// TIA Portal V19 export
FUNCTION "FC_FW_Auftrag_Step5_NB" : Void   // FC185, LAD
TITLE = Schritt CM04 -> WR02
{ S7_Optimized_Access := 'TRUE' }
// Ältesten Warenträger in CM04 suchen und nach WR02 transportieren
// stored: AutoNumber false, SetENOAutomatically false
   VAR_INPUT
      Frg_Schritt : Bool;
   END_VAR
   VAR_OUTPUT
      nextStep : Bool;
      startStep : Bool;
      parkStep : Bool;
   END_VAR
   VAR_IN_OUT
      Quelle : Int;
      Ziel : Int;
      Positionen : Array[1..30] of "UDT_Auftrag_Pos";
      Frg_Ausfahrt : Bool;
   END_VAR
   VAR_TEMP
      Sperre_Kurz_li : Bool;
      Sperre_Kurz_re : Bool;
      Sperre_Lang : Bool;
      Vorzug : Bool;
      Befehl_ok : Bool;
      tmpQuelle : Int;
      Oldest : Real;
   END_VAR
BEGIN

REGION Network 1 (SCL)
   IF (#Quelle <> 0) AND (#Ziel <> 0) THEN
       #nextStep := #Positionen[#Quelle].Sperre;
       #startStep := NOT #nextStep;
       #Quelle := 0;
       #Ziel := 0;
       #Frg_Ausfahrt := NOT #startStep;
       RETURN;
   END_IF;

   #Quelle := 0;
   #Ziel := 0;
   #nextStep := FALSE;
   #startStep := FALSE;
END_REGION

REGION Network 2 (SCL): Anmeldung Großoptik
   //alle Positionen suchbar
   #Positionen[19].CheckSperre := FALSE;
   #Positionen[20].CheckSperre := FALSE;
   #Positionen[21].CheckSperre := FALSE;
   #Positionen[22].CheckSperre := FALSE;
   #Positionen[23].CheckSperre := FALSE;
   #Positionen[24].CheckSperre := FALSE;

   //
   #Oldest := 0;
   #tmpQuelle := 0;

   //CM04
   "FC_FW_Auftrag_Suche"(Pos1 := 19,
                         Pos2 := 24,
                         Positionen := #Positionen,
                         Quelle := #tmpQuelle,
                         Oldest := #Oldest);

   IF ((#tmpQuelle = 21) OR (#tmpQuelle = 22)) AND #Frg_Ausfahrt AND #Frg_Schritt THEN
       //Großoptik ist ältester
       #Vorzug := NOT "DI_QF_WR02_03".In.Req_Ausfahrt_GO;
       "DI_QF_WR02_03".In.Req_Ausfahrt_GO := TRUE;
   ELSE
       #Vorzug := FALSE;
       "DI_QF_WR02_03".In.Req_Ausfahrt_GO := FALSE;
   END_IF;

   IF (#tmpQuelle = 0) OR NOT #Frg_Schritt THEN
       #Frg_Ausfahrt := FALSE;
   END_IF;
END_REGION

REGION Network 3 (SCL): Positionen sperren
   IF NOT #Frg_Ausfahrt OR NOT #Frg_Schritt THEN
       #nextStep := TRUE;
       RETURN;
   END_IF;

   //Groß links nicht möglich
   #Positionen[21].CheckSperre := #Positionen[27].Sperre;

   //Groß rechts nicht möglich
   #Positionen[22].CheckSperre := #Positionen[28].Sperre;

   //kein Platz für Kurz links in WR02
   #Sperre_Kurz_li := (#Positionen[25].Sperre AND #Positionen[29].Sperre) OR #Vorzug;

   //kein Platz für Kurz rechts in WR02
   #Sperre_Kurz_re := (#Positionen[26].Sperre AND #Positionen[30].Sperre) OR #Vorzug;

   //kein Platz für Lang in WR02
   #Sperre_Lang := ((#Positionen[25].Sperre OR #Positionen[26].Sperre) AND (#Positionen[29].Sperre OR #Positionen[30].Sperre)) OR #Vorzug;

   //Lang in P19 oder
   //kein Platz auf rechter Seite
   //-> P20 sperren
   #Positionen[20].CheckSperre := #Sperre_Kurz_re OR (#Positionen[19].Wt_Typ = "WT_Typ_LS");

   //Lang in P19 und kein Platz für Lang oder
   //kein Platz auf linker Seite
   //-> P19 sperren
   #Positionen[19].CheckSperre := #Sperre_Kurz_li OR ((#Positionen[19].Wt_Typ = "WT_Typ_LS") AND #Sperre_Lang);

   //Lang in P23 oder
   //kein Platz auf rechter Seite
   //-> P24 sperren
   #Positionen[24].CheckSperre := #Sperre_Kurz_re OR (#Positionen[23].Wt_Typ = "WT_Typ_LS");

   //Lang in P23 und kein Platz für Lang oder
   //kein Platz auf linker Seite
   //-> P23 sperren
   #Positionen[23].CheckSperre := #Sperre_Kurz_li OR ((#Positionen[23].Wt_Typ = "WT_Typ_LS") AND #Sperre_Lang);
END_REGION

REGION Network 4 (SCL): Ältesten WT suchen
   //
   #Oldest := 0;
   #tmpQuelle := 0;

   //CM04
   "FC_FW_Auftrag_Suche"(Pos1 := 19,
                         Pos2 := 24,
                         Positionen := #Positionen,
                         Quelle := #tmpQuelle,
                         Oldest := #Oldest);
END_REGION

REGION Network 5 (SCL): Auswertung
   IF #tmpQuelle = 0 THEN
       //kein WT
       #nextStep := TRUE;
       RETURN;
   END_IF;

   IF NOT #Positionen[#tmpQuelle].Fertig THEN
       #parkStep := TRUE;
       RETURN;
   END_IF;

   IF (#tmpQuelle = 21) THEN
       //Gross links
       IF NOT #Positionen[27].Sperre THEN
           "FC_FW_Auftrag_Befehl"(inQuelle := #tmpQuelle,
                                  inZiel := 27,
                                  Befehl_ok => #Befehl_ok,
                                  outQuelle => #Quelle,
                                  outZiel => #Ziel);

           #nextStep := NOT #Befehl_ok;
       ELSE
           #nextStep := TRUE;
       END_IF;
       RETURN;
   END_IF;

   IF (#tmpQuelle = 22) THEN
       //Gross rechts
       IF NOT #Positionen[28].Sperre THEN
           "FC_FW_Auftrag_Befehl"(inQuelle := #tmpQuelle,
                                  inZiel := 28,
                                  Befehl_ok => #Befehl_ok,
                                  outQuelle => #Quelle,
                                  outZiel => #Ziel);

           #nextStep := NOT #Befehl_ok;
       ELSE
           #nextStep := TRUE;
       END_IF;
       RETURN;
   END_IF;

   IF (#Positionen[#tmpQuelle].Wt_Typ = "WT_Typ_LS") AND ((#tmpQuelle = 19) OR (#tmpQuelle = 23)) THEN
       //Lang
       IF NOT #Positionen[25].Sperre AND NOT #Positionen[26].Sperre THEN
           "FC_FW_Auftrag_Befehl"(inQuelle := #tmpQuelle,
                                  inZiel := 25,
                                  Befehl_ok => #Befehl_ok,
                                  outQuelle => #Quelle,
                                  outZiel => #Ziel);

           #nextStep := NOT #Befehl_ok;
       ELSIF NOT #Positionen[29].Sperre AND NOT #Positionen[30].Sperre THEN
           "FC_FW_Auftrag_Befehl"(inQuelle := #tmpQuelle,
                                  inZiel := 29,
                                  Befehl_ok => #Befehl_ok,
                                  outQuelle => #Quelle,
                                  outZiel => #Ziel);

           #nextStep := NOT #Befehl_ok;
       ELSE
           #nextStep := TRUE;
       END_IF;
       RETURN;
   END_IF;

   IF (#tmpQuelle = 19) OR (#tmpQuelle = 23) THEN
       //Kurz links
       #Vorzug := NOT #Positionen[25].Sperre AND NOT #Positionen[26].Sperre AND NOT #Positionen[29].Sperre AND #Positionen[30].Sperre;

       IF NOT #Positionen[25].Sperre AND NOT #Vorzug THEN
           "FC_FW_Auftrag_Befehl"(inQuelle := #tmpQuelle,
                                  inZiel := 25,
                                  Befehl_ok => #Befehl_ok,
                                  outQuelle => #Quelle,
                                  outZiel => #Ziel);

           #nextStep := NOT #Befehl_ok;
       ELSIF NOT #Positionen[29].Sperre THEN
           "FC_FW_Auftrag_Befehl"(inQuelle := #tmpQuelle,
                                  inZiel := 29,
                                  Befehl_ok => #Befehl_ok,
                                  outQuelle => #Quelle,
                                  outZiel => #Ziel);

           #nextStep := NOT #Befehl_ok;
       ELSE
           #nextStep := TRUE;
       END_IF;
       RETURN;
   END_IF;

   IF (#tmpQuelle = 20) OR (#tmpQuelle = 24) THEN
       //Kurz rechts
       #Vorzug := NOT #Positionen[25].Sperre AND NOT #Positionen[26].Sperre AND #Positionen[29].Sperre AND NOT #Positionen[30].Sperre;

       IF NOT #Positionen[26].Sperre AND NOT #Vorzug THEN
           "FC_FW_Auftrag_Befehl"(inQuelle := #tmpQuelle,
                                  inZiel := 26,
                                  Befehl_ok => #Befehl_ok,
                                  outQuelle => #Quelle,
                                  outZiel => #Ziel);

           #nextStep := NOT #Befehl_ok;
       ELSIF NOT #Positionen[30].Sperre THEN
           "FC_FW_Auftrag_Befehl"(inQuelle := #tmpQuelle,
                                  inZiel := 30,
                                  Befehl_ok => #Befehl_ok,
                                  outQuelle => #Quelle,
                                  outZiel => #Ziel);

           #nextStep := NOT #Befehl_ok;
       ELSE
           #nextStep := TRUE;
       END_IF;
       RETURN;
   END_IF;

   //?
   #nextStep := TRUE;
END_REGION
END_FUNCTION
